FUNCTION_BLOCK FB_Cylinder_SingleSensor EXTENDS FB_CylinderBase
VAR_INPUT
END_VAR
VAR_OUTPUT
END_VAR
VAR
	fbSensor		: FB_Sensor;
	rtSensor		: R_TRIG;
END_VAR

METHOD HardwareUpdate : BOOL
VAR_INPUT
END_VAR
rtSensor(CLK := fbSensor.Active);

IF bExtendCommand AND rtSensor.Q THEN
	bExtendedFeedback := TRUE;
END_IF

IF bRetractCommand AND rtSensor.Q THEN
	bRetractedFeedback := TRUE;
END_IF

IF NOT fbSensor.Active THEN
	bExtendedFeedback 	:= FALSE;
	bRetractedFeedback 	:= FALSE;
END_IF
END_METHOD

END_FUNCTION_BLOCK

(* stored: Version 1.1.0.1, ProductVersion 3.1.4024.9
   POU FB_Cylinder_SingleSensor: Id {fb960eeb-30ec-488d-bfa9-d2b96eb8425d}, SpecialFunc None
   Folder 01_SUPER_Overrides: Id {a35187ca-eeeb-44b8-ac44-93c0be12975a}
   Method HardwareUpdate: Id {7bdfaebe-985b-4715-bcd7-3a9214ff83df} *)
